// TIA Portal V17 export
// export: Created 2025-08-05T09:36:01.213384Z, ExportSetting WithDefaults, DisplayName Totally Integrated Automation Portal, DisplayVersion V17, DisplayName TIA Portal Openness, DisplayVersion V17, DisplayName TIA Portal Version Control Interface, DisplayVersion V17, DisplayName SINAMICS Startdrive Advanced, DisplayVersion V17, DisplayName SINAMICS Startdrive G130, G150, S120, S150, SINAMICS MV, S210, DisplayVersion V17, DisplayName SINAMICS Startdrive G110M, G120, G120C, G120D, G120P, G115D, DisplayVersion V17, DisplayName STEP 7 Professional, DisplayVersion V17, DisplayName STEP 7 Safety, DisplayVersion V17, DisplayName WinCC Advanced, DisplayVersion V17
TYPE "typeKeyenceHmi"
// V01.00
// stored: IsFailsafeCompliant false
   STRUCT
      Input : Struct   // Data from HMI
         StartLaser : Bool;   // Start Markiervorgang / Start marking process
         StartDmcRenew : Bool;   // Start DMC erneuern / Start renewing DMC
         ResetLaser : Bool;   // Reset Laser / Reset laser
         ResetFinishState : Bool;   // Fertigmeldung zurücksetzen / Finished message reset
         MistCollectorTrigger : Bool;   // Absaugung triggern / Trigger exhaust system / Trigger exhaust
         TeachDistanceSensor : Bool;   // Abstandsensor teachen / Teach distance sensor
         CameraTrigger : Bool;   // Kamera triggern / Trigger camera
         OffsetDistSensorDistance : Real;   // Offsetwert zum Abnullen des Abstandsensors / Offset value for resetting the distance sensor
         OffsetDistSensorAngle : Real;   // Offsetwert zum Abnullen des Abstandsensors / Offset value for resetting the distance sensor
      END_STRUCT;
      Output : Struct   // Data to HMI
         ElementVisible : Struct
            ButtonStartLaser : Bool;
            ButtonStartRenew : Bool;
            ButtonReset : Bool;
            ButtonResetFinishState : Bool;
            ButtonTrigMistCollector : Bool;
            ButtonTeachDistanceSensor : Bool;
            ButtonTriggerCamera : Bool;
            LabelStringData : Bool;
            LabelDmc : Bool;
            LabelPrgNr : Bool;
            LabelErrorCode : Bool;
            LabelFocus : Bool;
            LabelDistance : Bool;
            LabelMarkingTime : Bool;
            TextboxDistanceOffset : Bool;
            ImageMistCollector : Bool;
            ImageReadResult : Bool;
         END_STRUCT;
         ElementEnable : Struct
            ButtonStartLaser : Bool;
            ButtonStartRenew : Bool;
            ButtonReset : Bool;
            ButtonResetFinishState : Bool;
            ButtonTrigMistCollector : Bool;
            ButtonTeachDistanceSensor : Bool;
            TextboxDistanceOffset : Bool;
         END_STRUCT;
         ElementActive : Struct
            ButtonStartLaser : Bool;
            ButtonStartRenew : Bool;
            ButtonReset : Bool;
            ButtonResetFinishState : Bool;
            ButtonTrigMistCollector : Bool;
            ButtonTeachDistanceSensor : Bool;
         END_STRUCT;
         Data : Struct
            Image : Struct   // Steuerung HMI Bilder / Control HMI screens
               LaserReady : Byte;   // Laser Betriebsbereit / Laser ready for operation
               LaserSelected : Byte;   // Markiereinheit aktiv / Marking unit active
               WorkpieceInPosition : Byte;   // Werstkück in Position / Part in position
               SafetyCircuit : Byte;   // Schutzkreis / Protective circuit
               Error : Byte;   // Störung / Fault / Failure
               KeySwitch : Byte;   // Schlüsselschalter / Key-operated switch
               MistCollector : Byte;   // Absaugung / Exhaust system / Exhaust
               Laser : Byte;   // Laser
               Shutter : Byte;   // Verschluss / Seal
               LaserFinished : Byte;   // Fertigmeldung Laser / Finished message laser
               StartMarking : Byte;   // Start Markieren / Start marking
               StartRenew : Byte;   // Start DMC Renew / Start DMC renew
               ResetLaser : Byte;   // Reset Laser / Reset laser
               quality : Byte;   // Leseergebnis / Qualität / Reset laser / Read result/quality
            END_STRUCT;
            LaserStatus : Struct
               TriggerReady : Bool;
               Error : Bool;
               Warning : Bool;
               Notice : Bool;
               Shutter : Bool;
               StartUp : Bool;
               res_0_6 : Bool;
               res_0_7 : Bool;
               Laser_Emit : Bool;
               ShutterControl : Bool;
               RemoteInterlock : Bool;
               Contacter : Bool;
               res_1_4 : Bool;
               res_1_5 : Bool;
               res_1_6 : Bool;
               res_1_7 : Bool;
               Busy : Bool;
               PrintBusy : Bool;
               GuidePrintBusy : Bool;
               ChangeBusy : Bool;
               LockBusy : Bool;
               EditBusy : Bool;
               Code2DReaderBusy : Bool;
               res_2_7 : Bool;
               res_3_0 : Bool;
               res_3_1 : Bool;
               res_3_2 : Bool;
               res_3_3 : Bool;
               res_3_4 : Bool;
               res_3_5 : Bool;
               res_3_6 : Bool;
               res_3_7 : Bool;
            END_STRUCT;
            ErrorCodeIntern : Int;   // interner Fehler Code / RESPONSE - VALUE 1 / Internal error code
            CharacterString : String[100];   // DMC Beschriftungsinhalt / DMC labeling content
            ReadDmc : String;   // gelesener DMC / Read DMC
            Status : Byte;   // aktueller Status / Current status
            CommandActive : Bool;   // Ablauf aktiv / Sequence active
            Offset : Struct   // Anzeige der hinterlegten Parameter Offsets / Display of stored parameter offsets
               Power : Real;   // aktueller Offset: Leistung / Current offset: power
               Frequence : Real;   // aktueller Offset: Frequenz / Current offset: frequency
               Speed : Real;   // aktueller Offset: Geschwindigkeit / Current offset: speed
               Defocus : Real;   // aktueller Offset: Defokus / Current offset: defocus
               Pulse_Width : Real;   // aktueller Offset: Pulsweite / Current offset: pulse width
            END_STRUCT;
            DistanceSensor : Struct   // Anzeige Abstandsensor / Display distance sensor
               Difference : Real;   // Differenz: Settingwert - Aktualwert / Difference: setting value - current value
               CurrentValue : Real;   // Aktualwert / Current value
               SettingValue : Real;   // Settingwert / Setting value
               Offset : Real;
            END_STRUCT;
            Zusatinformationen : Struct
               PrgNr : Array[1..4] of Char;   // Programmnummer / Loaded marking file / Program number
               ErrorCodesLaser : Array[1..3] of Int;   // Fehler Codes vom Laser / Error codes from the laser
               CommandError : Word;
               MarkingTime : Real;   // Beschriftungszeit - Markiervorgang / Labeling time - marking process
               TotalTime : Real;   // Beschriftungszeit - Gesamtablauf / Labeling time - complete cycle
               Length : Int;
               DataMatrix : Array[1..100] of Char;
            END_STRUCT;
         END_STRUCT;
      END_STRUCT;
   END_STRUCT;
END_TYPE
